// TIA Portal V18 export
FUNCTION_BLOCK "monitor_sw_no_encoder"   // FB36, FBD
{ S7_Optimized_Access := 'TRUE' }
VERSION : 0.1
// stored: AutoNumber true, IsIECCheckEnabled false, IsRetainMemResEnabled false, MemoryReserve 100, SetENOAutomatically false, UDAEnableTagReadback false
   VAR_INPUT
      xFWD : Bool;
      xFWDSLO : Bool;
      xREVSLO : Bool;
      xREV : Bool;
      go_FWD : Bool;
      go_REV : Bool;
      para_slo_to_slo : Time := T#2m;
      para_slo_to_end : Time := T#1m;
   END_VAR
   VAR_OUTPUT
      ER_FWD : Bool;
      ER_FWDSLO : Bool;
      ER_REVSLO : Bool;
      ER_REV : Bool;
   END_VAR
   VAR
      ton_fwd { S7_SetPoint := 'True'} : TON_TIME;
      ton_rev { S7_SetPoint := 'True'} : TON_TIME;
      ton_fwdslo { S7_SetPoint := 'True'} : TON_TIME;
      ton_revslo { S7_SetPoint := 'True'} : TON_TIME;
   END_VAR
BEGIN

REGION Network 1
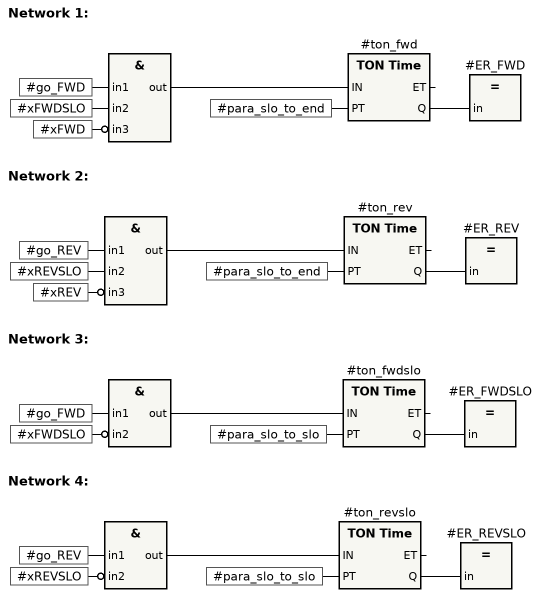
   #ton_fwd(IN := #go_FWD AND #xFWDSLO AND NOT #xFWD, PT := #para_slo_to_end);   // TON
   #ER_FWD := #ton_fwd.Q;
END_REGION

REGION Network 2
   #ton_rev(IN := #go_REV AND #xREVSLO AND NOT #xREV, PT := #para_slo_to_end);   // TON
   #ER_REV := #ton_rev.Q;
END_REGION

REGION Network 3
   #ton_fwdslo(IN := #go_FWD AND NOT #xFWDSLO, PT := #para_slo_to_slo);   // TON
   #ER_FWDSLO := #ton_fwdslo.Q;
END_REGION

REGION Network 4
   #ton_revslo(IN := #go_REV AND NOT #xREVSLO, PT := #para_slo_to_slo);   // TON
   #ER_REVSLO := #ton_revslo.Q;
END_REGION
END_FUNCTION_BLOCK
